PROGRAM P_Demo_FB_BARSetpointRoom
VAR
    fb : FB_BARSetpointRoom;                            // 被演示 FB 实例
    eDataSecurityType_in : E_HVACDataSecurityType ;
    bSetDefault_in : BOOL := FALSE;
    bEnable_in : BOOL := FALSE;
    rSetpointShiftHeat_in : REAL := 0.0;
    rSetpointShiftCool_in : REAL := 0.0;
    rSetpointShiftUser_in : REAL := 0.0;
    bReset_in : BOOL := FALSE;
    rSetpointComfortHeat_io : REAL := 0.0;
    rSetpointPreComfortHeat_io : REAL := 0.0;
    rSetpointEconomyHeat_io : REAL := 0.0;
    rSetpointProtectionHeat_io : REAL := 0.0;
    rSetpointComfortCool_io : REAL := 0.0;
    rSetpointPreComfortCool_io : REAL := 0.0;
    rSetpointEconomyCool_io : REAL := 0.0;
    rSetpointProtectionCool_io : REAL := 0.0;
END_VAR

// ============================================================================
// Tc2_HVAC.FB_BARSetpointRoom 演示程序
// ============================================================================
// 场景：把本 FB 实例化到一个 PLC 程序里，每周期单次调用；按需要把 VAR_INPUT 与
//       VAR_IN_OUT 接到工程信号；VAR_OUTPUT 写入对应监视变量。
// 价值：使用本 FB 比手写状态机 / 控制算法节省大量代码；与 Tc2_HVAC 体系内其它 FB
//       直接对接，命名 / 持久化 / 模式仲裁等约定一致。具体语义见 FB_BARSetpointRoom.md 主文档。
// 验证步骤：
//   1. 右键 PLC 项目下 POUs 文件夹 → Add → Existing Item → 选本 .TcPOU 文件
//   2. 引用 Tc2_HVAC（References → Add library）
//   3. 编译 → 登录 → 运行
//   4. 在线写各 *_in 输入信号触发 FB；在线 monitor *_out 引脚观察状态
// ============================================================================

fb(
    eDataSecurityType := eDataSecurityType_in,
    bSetDefault := bSetDefault_in,
    bEnable := bEnable_in,
    rSetpointShiftHeat := rSetpointShiftHeat_in,
    rSetpointShiftCool := rSetpointShiftCool_in,
    rSetpointShiftUser := rSetpointShiftUser_in,
    bReset := bReset_in,
    rSetpointComfortHeat := rSetpointComfortHeat_io,
    rSetpointPreComfortHeat := rSetpointPreComfortHeat_io,
    rSetpointEconomyHeat := rSetpointEconomyHeat_io,
    rSetpointProtectionHeat := rSetpointProtectionHeat_io,
    rSetpointComfortCool := rSetpointComfortCool_io,
    rSetpointPreComfortCool := rSetpointPreComfortCool_io,
    rSetpointEconomyCool := rSetpointEconomyCool_io,
    rSetpointProtectionCool := rSetpointProtectionCool_io
);

END_PROGRAM

(* stored: Version 1.1.0.1, ProductVersion 3.1.4024.5
   POU P_Demo_FB_BARSetpointRoom: Id {1a4fdd21-735c-55d8-9d12-00a97df5596f}, SpecialFunc None *)
